{attribute 'qualified_only'}
{attribute 'strict'}
TYPE E_Status :
(
	Ready,
	NotReady
);
END_TYPE

(* stored: Version 1.1.0.1, ProductVersion 3.1.4024.12
   DUT E_Status: Id {cdc7febb-de83-4c38-bc0f-470eb5f190fc} *)
